ABB RobotStudio station: ProyectoRobotica.rspag

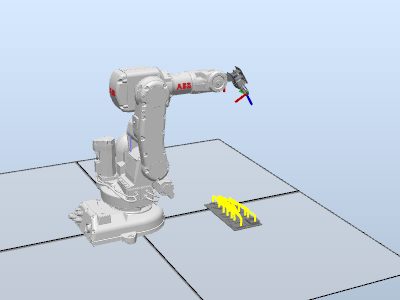
--- station ---
Station ProyectoRobotica (saved by RobotStudio 22.2.9947.0)
Controller ProyectoRobotica
  mechanical unit ROB_1: IRB140_6_81_C_03, 6 joints, base frame (0, 0, 0) mm
Layout (positions relative to the parent item):
  - IRB140_6_81_C_03 [mechanism, from Robots\IRB140_6_81_C_G_03.rslib] at (0, 0, 0) mm; joint values [0, 0, 0, 0, 0, 0.0001] (rad or m)
  - Gripper_Tool [part] at (577.08, 0, 697.04) mm, rotated rx 0 ry -30 rz 0 deg, size 101.4 x 78.8 x 170.9 mm
  - BaseEns [part] at (550, 0, 5) mm, rotated rx 180 ry 0 rz 90 deg, size 350 x 160 x 30 mm
  - PestCent [part] at (578.58, -114.16, 9) mm, rotated rx 0 ry 90 rz 0 deg, size 4 x 21.7 x 39.9 mm
  - Corto [part] at (540.6, -47.6, 7.04) mm, rotated rx 0 ry 90 rz 39 deg, size 4 x 17.8 x 15.7 mm
  - Corto_2 [part] at (473.4, -179, 7.04) mm, rotated rx 0 ry 90 rz -141 deg, size 4 x 17.8 x 15.7 mm
  - Punta [part] at (551.4, -103.2, 13) mm, rotated rx 0 ry 90 rz 0 deg, size 6 x 18.2 x 33.2 mm
  - Punta_2 [part] at (551.4, -123.4, 3) mm, rotated rx 0 ry -90 rz -180 deg, size 6 x 18.2 x 33.2 mm
  - Tapa1 [part] at (565, -250, 5) mm, rotated rx 0 ry -90 rz -180 deg, size 16 x 60 x 70 mm
  - Tapa2 [part] at (485, -250, 9) mm, rotated rx 0 ry -90 rz -180 deg, size 8 x 60 x 70 mm
  - Largo [part] at (534, -169.47, 9) mm, rotated rx 0 ry 90 rz 24.7 deg, size 4 x 24.5 x 44.3 mm
  - Largo_2 [part] at (534, -197.47, 9) mm, rotated rx 0 ry 90 rz 24.7 deg, size 4 x 24.5 x 44.3 mm
  - Largo_3 [part] at (613.2, -169.47, 9) mm, rotated rx 0 ry 90 rz 24.7 deg, size 4 x 24.5 x 44.3 mm
  - Largo_4 [part] at (613.4, -197.47, 9) mm, rotated rx 0 ry 90 rz 24.7 deg, size 4 x 24.5 x 44.3 mm
  - MontajeGripperFinal [part] at (464.9, -30.3, -4.6) mm, rotated rx 90 ry 0 rz 90 deg, size 92.4 x 24 x 121.8 mm
Attachment: Gripper_Tool is attached to IRB140_6_81_C_03 / Link6

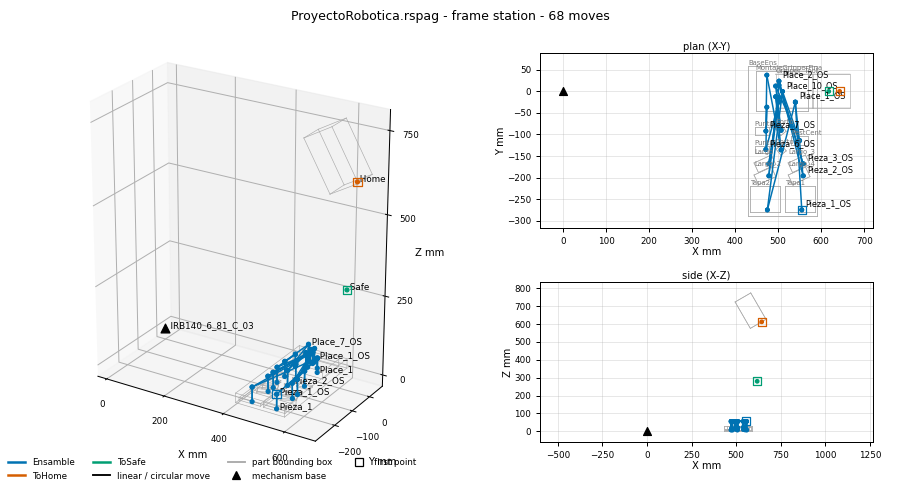
[picture p0: tool path of ProyectoRobotica.rspag in frame station, 68 of 68 moves have a stored position in this frame; points joined in program order, loops and branches not executed]
--- Controller Data/ProyectoRobotica/RAPID/TASK1/PROGMOD/CalibData.mod ---
MODULE CalibData
    TASK PERS tooldata GripperTool:=[TRUE,[[99,0,128],[0.866025404,0,0.5,0]],[1,[0,0,1],[1,0,0,0],0,0,0]];
    TASK PERS wobjdata Tabla:=[FALSE,TRUE,"",[[374.761,459.614,5],[0.38267537,0,0,0.923882872]],[[-434.758626611,130.385884139,0],[0.923879533,0,0,-0.382683431]]];
ENDMODULE

--- Controller Data/ProyectoRobotica/RAPID/TASK1/PROGMOD/Module1.mod ---
MODULE Module1
    CONST robtarget Pieza_1_OS:=[[-335,35,50],[0,0.707106781,0.707106781,0],[-1,-1,0,1],[9E+09,9E+09,9E+09,9E+09,9E+09,9E+09]];
    CONST robtarget Pieza_1:=[[-335,35,4],[0,0.707106781,0.707106781,0],[-1,-1,0,1],[9E+09,9E+09,9E+09,9E+09,9E+09,9E+09]];
    CONST robtarget Place_1_OS:=[[-85,50,50],[0,0.707106781,0.707106781,0],[-1,-1,0,1],[9E+09,9E+09,9E+09,9E+09,9E+09,9E+09]];
    CONST robtarget Place_1:=[[-85,50,4],[0,0.707106781,0.707106781,0],[-1,-1,0,1],[9E+09,9E+09,9E+09,9E+09,9E+09,9E+09]];
    CONST robtarget Pieza_2_OS:=[[-256,32,50],[0,0.707106781,0.707106781,0],[-1,-1,0,1],[9E+09,9E+09,9E+09,9E+09,9E+09,9E+09]];
    CONST robtarget Pieza_2:=[[-256,31,2],[0,0.707106781,0.707106781,0],[-1,-1,0,1],[9E+09,9E+09,9E+09,9E+09,9E+09,9E+09]];
    CONST robtarget Place_2_OS:=[[-36.132,88,50],[0,0.898794046,0.438371147,0],[0,0,-1,1],[9E+09,9E+09,9E+09,9E+09,9E+09,9E+09]];
    CONST robtarget Place_2:=[[-36.132,88,6],[0,0.898794046,0.438371147,0],[0,0,-1,1],[9E+09,9E+09,9E+09,9E+09,9E+09,9E+09]];
    CONST robtarget Pieza_3_OS:=[[-228,32,50],[0,0.707106781,0.707106781,0],[-1,-1,0,1],[9E+09,9E+09,9E+09,9E+09,9E+09,9E+09]];
    CONST robtarget Pieza_3:=[[-228,31,2],[0,0.707106781,0.707106781,0],[-1,-1,0,1],[9E+09,9E+09,9E+09,9E+09,9E+09,9E+09]];
    CONST robtarget Place_3_OS:=[[-45.774,88,50],[0,0.898794046,0.438371147,0],[0,0,-1,1],[9E+09,9E+09,9E+09,9E+09,9E+09,9E+09]];
    CONST robtarget Place_3:=[[-45.774,88,10],[0,0.898794046,0.438371147,0],[0,0,-1,1],[9E+09,9E+09,9E+09,9E+09,9E+09,9E+09]];
    CONST robtarget Pieza_4_OS:=[[-256,111.667,50],[0,0.707106781,0.707106781,0],[-1,-1,0,1],[9E+09,9E+09,9E+09,9E+09,9E+09,9E+09]];
    CONST robtarget Pieza_4:=[[-256,110.667,2],[0,0.707106781,0.707106781,0],[-1,-1,0,1],[9E+09,9E+09,9E+09,9E+09,9E+09,9E+09]];
    CONST robtarget Place_4_OS:=[[-74.431,88,50],[0,0.469471563,0.882947593,0],[-1,-1,0,1],[9E+09,9E+09,9E+09,9E+09,9E+09,9E+09]];
    CONST robtarget Place_4:=[[-74.431,88,6],[0,0.469471561,0.882947594,0],[-1,-1,0,1],[9E+09,9E+09,9E+09,9E+09,9E+09,9E+09]];
    CONST robtarget Pieza_5_OS:=[[-228,111.667,50],[0,0.707106781,0.707106781,0],[-1,-1,0,1],[9E+09,9E+09,9E+09,9E+09,9E+09,9E+09]];
    CONST robtarget Pieza_5:=[[-228,110.667,2],[0,0.707106781,0.707106781,0],[-1,-1,0,1],[9E+09,9E+09,9E+09,9E+09,9E+09,9E+09]];
    CONST robtarget Place_5_OS:=[[-84.431,88,50],[0,0.469471563,0.882947593,0],[-1,-1,0,1],[9E+09,9E+09,9E+09,9E+09,9E+09,9E+09]];
    CONST robtarget Place_5:=[[-84.431,88,10],[0,0.469471563,0.882947593,0],[-1,-1,0,1],[9E+09,9E+09,9E+09,9E+09,9E+09,9E+09]];
    CONST robtarget Pieza_6_OS:=[[-194.858,118.467,50],[0,0.707106781,0.707106781,0],[-1,-1,0,1],[9E+09,9E+09,9E+09,9E+09,9E+09,9E+09]];
    CONST robtarget Pieza_6:=[[-194.858,118.467,2],[0,0.707106781,0.707106781,0],[-1,-1,0,1],[9E+09,9E+09,9E+09,9E+09,9E+09,9E+09]];
    CONST robtarget Place_6_OS:=[[-96.61,116.228,50],[0,0.707106781,0.707106781,0],[-1,-1,0,1],[9E+09,9E+09,9E+09,9E+09,9E+09,9E+09]];
    CONST robtarget Place_6:=[[-96.61,116.228,10],[0,0.707106781,0.707106781,0],[-1,-1,0,1],[9E+09,9E+09,9E+09,9E+09,9E+09,9E+09]];
    CONST robtarget Pieza_7_OS:=[[-152.082,118.467,50],[0,0.707106781,0.707106781,0],[-1,-1,0,1],[9E+09,9E+09,9E+09,9E+09,9E+09,9E+09]];
    CONST robtarget Pieza_7:=[[-152.082,118.467,2],[0,0.707106781,0.707106781,0],[-1,-1,0,1],[9E+09,9E+09,9E+09,9E+09,9E+09,9E+09]];
    CONST robtarget Place_7_OS:=[[-22.317,116.228,50],[0,0.707106781,0.707106781,0],[0,0,-1,1],[9E+09,9E+09,9E+09,9E+09,9E+09,9E+09]];
    CONST robtarget Place_7:=[[-22.317,116.228,10],[0,0.707106781,0.707106781,0],[0,0,-1,1],[9E+09,9E+09,9E+09,9E+09,9E+09,9E+09]];
    CONST robtarget Pieza_8_OS:=[[-195.858,82.967,50],[0,1,0,0],[-1,1,-1,1],[9E+09,9E+09,9E+09,9E+09,9E+09,9E+09]];
    CONST robtarget Pieza_8:=[[-195.858,82.967,2],[0,1,0,0],[-1,1,-1,1],[9E+09,9E+09,9E+09,9E+09,9E+09,9E+09]];
    CONST robtarget Place_8_OS:=[[-72.342,95.74,50],[0,1,0,0],[0,1,-1,1],[9E+09,9E+09,9E+09,9E+09,9E+09,9E+09]];
    CONST robtarget Place_8:=[[-72.342,95.74,10],[0,1,0,0],[0,1,-1,1],[9E+09,9E+09,9E+09,9E+09,9E+09,9E+09]];
    CONST robtarget Pieza_9_OS:=[[-150.322,82.967,50],[0,1,0,0],[0,1,-1,1],[9E+09,9E+09,9E+09,9E+09,9E+09,9E+09]];
    CONST robtarget Pieza_9:=[[-150.322,82.967,2],[0,1,0,0],[0,1,-1,1],[9E+09,9E+09,9E+09,9E+09,9E+09,9E+09]];
    CONST robtarget Place_9_OS:=[[-47.65,95.74,50],[0,1,0,0],[0,1,-1,1],[9E+09,9E+09,9E+09,9E+09,9E+09,9E+09]];
    CONST robtarget Place_9:=[[-47.65,95.74,10],[0,1,0,0],[0,1,-1,1],[9E+09,9E+09,9E+09,9E+09,9E+09,9E+09]];
    CONST robtarget Pieza_10_OS:=[[-174.155,39.9,50],[0,1,0,0],[0,1,-1,1],[9E+09,9E+09,9E+09,9E+09,9E+09,9E+09]];
    CONST robtarget Pieza_10:=[[-174.155,39.9,2],[0,1,0,0],[0,1,-1,1],[9E+09,9E+09,9E+09,9E+09,9E+09,9E+09]];
    CONST robtarget Place_10_OS:=[[-60,79.85,50],[0,1,0,0],[0,1,-1,1],[9E+09,9E+09,9E+09,9E+09,9E+09,9E+09]];
    CONST robtarget Place_10:=[[-60,79.85,14],[0,1,0,0],[0,1,-1,1],[9E+09,9E+09,9E+09,9E+09,9E+09,9E+09]];
    CONST robtarget Pieza_11_OS:=[[-335,115,50],[0,0.707106781,0.707106781,0],[-1,-1,0,1],[9E+09,9E+09,9E+09,9E+09,9E+09,9E+09]];
    CONST robtarget Pieza_11:=[[-335,115,4],[0,0.707106781,0.707106781,0],[-1,-1,0,1],[9E+09,9E+09,9E+09,9E+09,9E+09,9E+09]];
    CONST robtarget Place_11_OS:=[[-85,50,50],[0,0.707106781,0.707106781,0],[-1,-1,0,1],[9E+09,9E+09,9E+09,9E+09,9E+09,9E+09]];
    CONST robtarget Place_11:=[[-85,50,18],[0,0.707106781,0.707106781,0],[-1,-1,0,1],[9E+09,9E+09,9E+09,9E+09,9E+09,9E+09]];
    CONST robtarget Home:=[[-59.995408426,-53.012265309,608.010207808],[0.183047251,0.683018555,0.682997169,-0.183014276],[0,0,0,0],[9E+09,9E+09,9E+09,9E+09,9E+09,9E+09]];
    CONST robtarget Safe:=[[-60.000216702,-27.649874409,274.763485025],[0,0.707112843,0.70710072,0],[0,0,-1,1],[9E+09,9E+09,9E+09,9E+09,9E+09,9E+09]];

    PROC main()
        WaitDI DI_01,1;
        SetDO DO_03,0;        !!Operando
        ToHome;
        ToSafe;
        Ensamble;
        ToSafe;
        ToHome;
        SetDO DO_03,1;        !!Fin
    ENDPROC

    PROC Ensamble()
        MoveJ Pieza_1_OS,v50,z5,GripperTool\WObj:=Tabla;
        WaitDI DI_02,1;
        MoveL Pieza_1,v10,z0,GripperTool\WObj:=Tabla;
        SetDO DO_01,1;
        WaitTime 2;
        SetDO DO_01,0;
        MoveL Pieza_1_OS,v10,z0,GripperTool\WObj:=Tabla;
        MoveL Place_1_OS,v50,z5,GripperTool\WObj:=Tabla;
        WaitDI DI_02,1;
        MoveL Place_1,v10,z0,GripperTool\WObj:=Tabla;
        SetDO DO_02,1;
        WaitTime 2;
        SetDO DO_02,0;
        MoveL Place_1_OS,v10,z0,GripperTool\WObj:=Tabla;
        MoveL Pieza_2_OS,v50,z5,GripperTool\WObj:=Tabla;
        WaitDI DI_02,1;
        MoveL Pieza_2,v10,z0,GripperTool\WObj:=Tabla;
        SetDO DO_01,1;
        WaitTime 2;
        SetDO DO_01,0;
        MoveL Pieza_2_OS,v10,z0,GripperTool\WObj:=Tabla;
        MoveL Place_2_OS,v50,z5,GripperTool\WObj:=Tabla;
        WaitDI DI_02,1;
        MoveL Place_2,v10,z0,GripperTool\WObj:=Tabla;
        SetDO DO_02,1;
        WaitTime 2;
        SetDO DO_02,0;
        MoveL Place_2_OS,v10,z0,GripperTool\WObj:=Tabla;
        MoveL Pieza_3_OS,v50,z5,GripperTool\WObj:=Tabla;
        WaitDI DI_02,1;
        MoveL Pieza_3,v10,z0,GripperTool\WObj:=Tabla;
        SetDO DO_01,1;
        WaitTime 2;
        SetDO DO_01,0;
        MoveL Pieza_3_OS,v10,z0,GripperTool\WObj:=Tabla;
        MoveL Place_3_OS,v50,z5,GripperTool\WObj:=Tabla;
        WaitDI DI_02,1;
        MoveL Place_3,v10,z0,GripperTool\WObj:=Tabla;
        SetDO DO_02,1;
        WaitTime 2;
        SetDO DO_02,0;
        MoveL Place_3_OS,v10,z0,GripperTool\WObj:=Tabla;
        MoveL Pieza_4_OS,v50,z5,GripperTool\WObj:=Tabla;
        WaitDI DI_02,1;
        MoveL Pieza_4,v10,z0,GripperTool\WObj:=Tabla;
        SetDO DO_01,1;
        WaitTime 2;
        SetDO DO_01,0;
        MoveL Pieza_4_OS,v10,z0,GripperTool\WObj:=Tabla;
        MoveL Place_4_OS,v50,z5,GripperTool\WObj:=Tabla;
        WaitDI DI_02,1;
        MoveL Place_4,v10,z0,GripperTool\WObj:=Tabla;
        SetDO DO_02,1;
        WaitTime 2;
        SetDO DO_02,0;
        MoveL Place_4_OS,v10,z0,GripperTool\WObj:=Tabla;
        MoveL Pieza_5_OS,v50,z5,GripperTool\WObj:=Tabla;
        WaitDI DI_02,1;
        MoveL Pieza_5,v10,z0,GripperTool\WObj:=Tabla;
        SetDO DO_01,1;
        WaitTime 2;
        SetDO DO_01,0;
        MoveL Pieza_5_OS,v10,z0,GripperTool\WObj:=Tabla;
        MoveL Place_5_OS,v50,z5,GripperTool\WObj:=Tabla;
        WaitDI DI_02,1;
        MoveL Place_5,v10,z0,GripperTool\WObj:=Tabla;
        SetDO DO_02,1;
        WaitTime 2;
        SetDO DO_02,0;
        MoveL Place_5_OS,v10,z0,GripperTool\WObj:=Tabla;
        MoveL Pieza_6_OS,v50,z5,GripperTool\WObj:=Tabla;
        WaitDI DI_02,1;
        MoveL Pieza_6,v10,z0,GripperTool\WObj:=Tabla;
        SetDO DO_01,1;
        WaitTime 2;
        SetDO DO_01,0;
        MoveL Pieza_6_OS,v10,z0,GripperTool\WObj:=Tabla;
        MoveL Place_6_OS,v50,z5,GripperTool\WObj:=Tabla;
        WaitDI DI_02,1;
        MoveL Place_6,v10,z0,GripperTool\WObj:=Tabla;
        SetDO DO_02,1;
        WaitTime 2;
        SetDO DO_02,0;
        MoveL Place_6_OS,v10,z0,GripperTool\WObj:=Tabla;
        MoveL Pieza_7_OS,v50,z5,GripperTool\WObj:=Tabla;
        WaitDI DI_02,1;
        MoveL Pieza_7,v10,z0,GripperTool\WObj:=Tabla;
        SetDO DO_01,1;
        WaitTime 2;
        SetDO DO_01,0;
        MoveL Pieza_7_OS,v10,z0,GripperTool\WObj:=Tabla;
        MoveL Place_7_OS,v50,z5,GripperTool\WObj:=Tabla;
        WaitDI DI_02,1;
        MoveL Place_7,v10,z0,GripperTool\WObj:=Tabla;
        SetDO DO_02,1;
        WaitTime 2;
        SetDO DO_02,0;
        MoveL Place_7_OS,v10,z0,GripperTool\WObj:=Tabla;
        MoveL Pieza_8_OS,v50,z5,GripperTool\WObj:=Tabla;
        WaitDI DI_02,1;
        MoveL Pieza_8,v10,z0,GripperTool\WObj:=Tabla;
        SetDO DO_01,1;
        WaitTime 2;
        SetDO DO_01,0;
        MoveL Pieza_8_OS,v10,z0,GripperTool\WObj:=Tabla;
        MoveL Place_8_OS,v50,z5,GripperTool\WObj:=Tabla;
        WaitDI DI_02,1;
        MoveL Place_8,v10,z0,GripperTool\WObj:=Tabla;
        SetDO DO_02,1;
        WaitTime 2;
        SetDO DO_02,0;
        MoveL Place_8_OS,v10,z0,GripperTool\WObj:=Tabla;
        MoveL Pieza_9_OS,v50,z5,GripperTool\WObj:=Tabla;
        WaitDI DI_02,1;
        MoveL Pieza_9,v10,z0,GripperTool\WObj:=Tabla;
        SetDO DO_01,1;
        WaitTime 2;
        SetDO DO_01,0;
        MoveL Pieza_9_OS,v10,z0,GripperTool\WObj:=Tabla;
        MoveL Place_9_OS,v50,z5,GripperTool\WObj:=Tabla;
        WaitDI DI_02,1;
        MoveL Place_9,v10,z0,GripperTool\WObj:=Tabla;
        SetDO DO_02,1;
        WaitTime 2;
        SetDO DO_02,0;
        MoveL Place_9_OS,v10,z0,GripperTool\WObj:=Tabla;
        MoveL Pieza_10_OS,v50,z5,GripperTool\WObj:=Tabla;
        WaitDI DI_02,1;
        MoveL Pieza_10,v10,z0,GripperTool\WObj:=Tabla;
        SetDO DO_01,1;
        WaitTime 2;
        SetDO DO_01,0;
        MoveL Pieza_10_OS,v10,z0,GripperTool\WObj:=Tabla;
        MoveL Place_10_OS,v50,z5,GripperTool\WObj:=Tabla;
        WaitDI DI_02,1;
        MoveL Place_10,v10,z0,GripperTool\WObj:=Tabla;
        SetDO DO_02,1;
        WaitTime 2;
        SetDO DO_02,0;
        MoveL Place_10_OS,v10,z0,GripperTool\WObj:=Tabla;
        MoveL Pieza_11_OS,v50,z5,GripperTool\WObj:=Tabla;
        WaitDI DI_02,1;
        MoveL Pieza_11,v10,z0,GripperTool\WObj:=Tabla;
        SetDO DO_01,1;
        WaitTime 2;
        SetDO DO_01,0;
        MoveL Pieza_11_OS,v10,z0,GripperTool\WObj:=Tabla;
        MoveL Place_11_OS,v50,z5,GripperTool\WObj:=Tabla;
        WaitDI DI_02,1;
        MoveL Place_11,v10,z0,GripperTool\WObj:=Tabla;
        SetDO DO_02,1;
        WaitTime 2;
        SetDO DO_02,0;
        MoveL Place_11_OS,v10,z0,GripperTool\WObj:=Tabla;
    ENDPROC
    PROC ToHome()
        MoveJ Home,v1000,z100,GripperTool\WObj:=Tabla;
    ENDPROC
    PROC ToSafe()
        MoveJ Safe,v100,z10,GripperTool\WObj:=Tabla;
    ENDPROC
ENDMODULE

--- Controller Data/ProyectoRobotica/SYSPAR/EIO.cfg ---
EIO:CFG_1.0:6:1::
#
EIO_SIGNAL:

      -Name "DO_01" -SignalType "DO" -Access "All"

      -Name "DO_02" -SignalType "DO" -Access "All"

      -Name "DO_03" -SignalType "DO" -Access "All"

      -Name "DI_01" -SignalType "DI" -Access "All"

      -Name "DI_02" -SignalType "DI" -Access "All"
